FUNCTION_BLOCK FB_Alarm EXTENDS FB_AlarmBase
VAR_INPUT
	bEnable				: BOOL;
END_VAR

bActive := bEnable;

SUPER^();

PROPERTY ArgStackMemoryPointer : POINTER TO BYTE
GET
ArgStackMemoryPointer := 0;
END_GET
END_PROPERTY

PROPERTY ArgStackMemorySize : DINT
GET
ArgStackMemorySize := 0;
END_GET
END_PROPERTY

METHOD PROTECTED  ClearArgStack
VAR_INPUT
END_VAR
// Do nothing
END_METHOD

METHOD PROTECTED CopyArgsToStack
VAR_INPUT
END_VAR
// Do nothing
END_METHOD

END_FUNCTION_BLOCK

(* stored: Version 1.1.0.1, ProductVersion 3.1.4024.15
   POU FB_Alarm: Id {cd7d921d-0cdd-4afc-8993-e9236f1ce3b5}, SpecialFunc None
   Property ArgStackMemoryPointer: Id {525c97dd-552f-4af1-8b84-cc7a352d131d}
   Get Get: Id {32102f1a-8ead-4711-ba95-0849989a0837}
   Property ArgStackMemorySize: Id {f05d1709-c924-4dce-bd0a-6bc6e39aef02}
   Get Get: Id {0e2403c8-7e80-4a45-812a-245642e865a7}
   Method ClearArgStack: Id {e19c0412-1b71-46c0-8417-7443def4245b}
   Method CopyArgsToStack: Id {66d5f472-79b2-4d41-803a-d0e0ed4c405c} *)
